PROGRAM Index_and_Measure
VAR
	RequestedRibLength:REAL; // Length in inches needed for ribs to cut
	MinRibLength: DINT; // Minimnm length of leftover that can still be used.
	MaxRibLength: DINT; // Longest rib lenght
	NumOfRibs:INT; // Quantity of tibs needed for next part
	RibRequest:BOOL; // Ribs needed for next part.
	RemainingLength:DINT; // Left over length of rib after cut
	PPI:REAL; // Pulses Per Inch from encoder
	CutLength: REAL; // Rib length to cut in encoder pulses 
	KerfWidth : REAL; // Width of saw blade in encoder pulses
	TotalCutLength : REAL; // Cut length requested plus kerf width of saw blade
	RibReadyToCut: BOOL; // Rib is in position to begin cutting
	HMI_PB_ManualJogFwd:BOOL; // HMI manual jog forward
	HMI_PB_ManualJogRev: bool; // HMI manual jog reverse
	IndexFwd: BOOL; // Clear path signal to go forward direction
	IndexRev: BOOL; // Clear path signal to go reverse direction
	OpenTransferClampRequest: BOOL;
	CloseTransferClampRequest: BOOL;
END_VAR

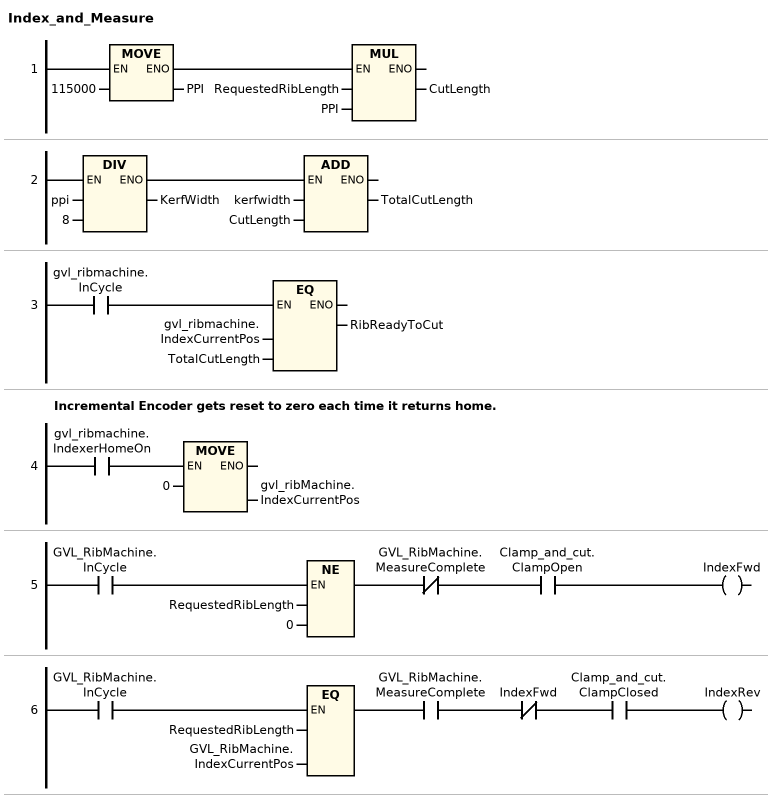
// NETWORK 1
PPI := 115000;
CutLength := RequestedRibLength * PPI;

// NETWORK 2
KerfWidth := ppi / 8;
TotalCutLength := kerfwidth + CutLength;

// NETWORK 3
IF gvl_ribmachine.InCycle THEN RibReadyToCut := gvl_ribmachine.IndexCurrentPos = TotalCutLength; END_IF

// NETWORK 4: Incremental Encoder gets reset to zero each time it returns home.
IF gvl_ribmachine.IndexerHomeOn THEN gvl_ribMachine.IndexCurrentPos := 0; END_IF

// NETWORK 5
IndexFwd := (GVL_RibMachine.InCycle AND RequestedRibLength <> 0) AND NOT GVL_RibMachine.MeasureComplete AND Clamp_and_cut.ClampOpen;

// NETWORK 6
IndexRev := (GVL_RibMachine.InCycle AND RequestedRibLength = GVL_RibMachine.IndexCurrentPos) AND GVL_RibMachine.MeasureComplete AND NOT IndexFwd AND Clamp_and_cut.ClampClosed;

END_PROGRAM

(* stored: Version 1.1.0.1, ProductVersion 3.1.4024.12
   POU Index_and_Measure: Id {968e1330-3aa7-4c4a-ae3b-4397f473161c}, SpecialFunc None *)
